PROGRAM P_Demo_F_BA_OffsetPtr
VAR
    argPAddr                       : PVOID                          := 0; // pAddr
    argNOffset                     : DINT                           := 0; // nOffset
    fnReturn                       : PVOID; // 返回值
END_VAR

// =============================================================================
// Tc3_BA2_Common.F_BA_OffsetPtr 演示程序
// =============================================================================
// 场景：操作 RAW 数据缓冲（如总线帧）：拿到帧头指针后 +4 跳过 header 取 payload 指针。
//
// 价值：跨 x86/x64 平台自动正确；手写 `pAddr + UDINT(nOffset)` 在 x64 上会把指针截断到 32 位 → 段错误。
//
// 验证：登录 PLC 后，按例程内变量在线写值；监视输出 / 返回值，结合 §1 功能
//       简述的预期行为对照（详见配套 .md 文档 §7 业务场景）。
//
// 验证步骤：
//   1. 右键 PLC 项目下 POUs 文件夹 → Add → Existing Item → 选本 .TcPOU 文件
//   2. 引用 Tc3_BA2_Common（References → Add library）
//   3. 编译 → 登录 → 运行；按上方『验证』指引在线写值观察
// =============================================================================

fnReturn := F_BA_OffsetPtr(
    pAddr                    := argPAddr,
    nOffset                  := argNOffset
);

END_PROGRAM

(* stored: Version 1.1.0.1, ProductVersion 3.1.4024.5
   POU P_Demo_F_BA_OffsetPtr: Id {fe484b58-4447-5735-ab33-29b92d92d2fc}, SpecialFunc None *)
